Omron CX-Programmer project NewProject (CX-Programmer 9.61)

# PLC NewPLC1: CP1E N30

## Global symbols (name address type ; comment)
0.00 BOOL  ; PB1
0.01 BOOL  ; S1
0.02 BOOL  ; PS1
0.03 BOOL  ; TS1
0.04 BOOL  ; S2
0.05 BOOL  ; S3
100.00 BOOL  ; L1

## Program NewProgram1 (cyclic task 0)

### Section Section1

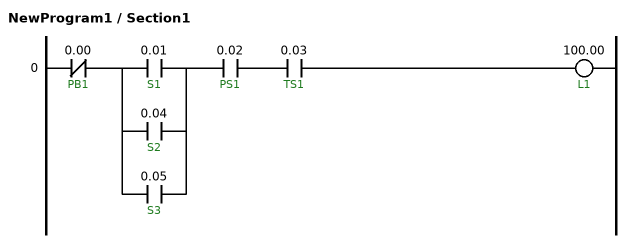
; rung 0
LDNOT 0.00  ; PB1
LD 0.01  ; S1
OR 0.04  ; S2
OR 0.05  ; S3
ANDLD
AND 0.02  ; PS1
AND 0.03  ; TS1
OUT 100.00  ; L1

### Section END
; rung 0
END(001)